(* CODESYS project Task1.project
   CompiledLibraryCompatibilityVersion: LeadSysStudio V3.5 SP15 Patch 4
   Title: Task1

Project tree, tasks and I/O mapping:
  Device : PMC600, Leadshine Technology Co., Ltd., order no. 600101, version 3.5.15.40
    application Application
      libraries: Standard, * (System)
      task MainTask (cyclic, interval t#4ms, priority 4, watchdog t#5000ms x 1) calls nothing
      task EtherCAT_Master_Leadshine_A (cyclic, interval 4000 µs, priority 0) calls PLC_PRG, EtherCAT_Master_Leadshine_A.EtherCAT_Task
      task SoftMotion_PlanningTask (freewheeling, priority 15) calls nothing
      program PLC_PRG [LD]
      axis group Tripod: TRAFO.Kin_Tripod_Rotary, axes Axis_3, Axis_4, Axis_5
    Device Diagnose
    Network Configuration
      LocalBus Config
    Resource Usage
    SoftMotion General Axis Pool
    High_Speed_IO_Module : High Speed IO Module, Leadshine Technology Co., Ltd., version 3.5.15.40
        unmapped channels: Genral_IO_IN, Genral_IO_Out
    EtherCAT_Master_Leadshine_A : EtherCAT Master Leadshine, Leadshine Technology Co., Ltd., version 3.5.9.50
        settings: MasterCycleTime = 4000
      PM32EC_LOCAL : PM32EC-LOCAL, Leadshine Technology Co., Ltd., order no. PM32EC-LOCAL, version Revision=16#20061010
          settings: StationAlias = 0; DC sync0 cycletime = 4000; DC sync1 cycletime = 4000
      DM3C_EC522 : DM3C-EC522(COE), Leadshine Technology Co.,Ltd., order no. DM3C-EC522, version Revision=16#00000001
          settings: StationAlias = 0; DC sync0 cycletime = 4000; DC sync1 cycletime = 4000; Number of SDO = 6; Homing method.Index = 16#6098; Homing method.Subindex = 16#00; Homing method.Value = 29; Homing method.Size = 8; Homing method.AbortIfError = FALSE; Homing method.JumpToLine = FALSE; Homing method.Line = 0; Homing method.CompleteAccess = FALSE; Homing velocity (fast).Index = 16#6099; Homing velocity (fast).Subindex = 16#01; Homing velocity (fast).Value = 1667; Homing velocity (fast).Size = 32; Homing velocity (fast).AbortIfError = FALSE; Homing velocity (fast).JumpToLine = FALSE; Homing velocity (fast).Line = 0; Homing velocity (fast).CompleteAccess = FALSE; Homing velocity (slow).Index = 16#6099; Homing velocity (slow).Subindex = 16#02; Homing velocity (slow).Value = 333; Homing velocity (slow).Size = 32; Homing velocity (slow).AbortIfError = FALSE; Homing velocity (slow).JumpToLine = FALSE; Homing velocity (slow).Line = 0; Homing velocity (slow).CompleteAccess = FALSE; Homing acceleration.Index = 16#609A; Homing acceleration.Subindex = 16#00; Homing acceleration.Value = 16667; Homing acceleration.Size = 32; Homing acceleration.AbortIfError = FALSE; Homing acceleration.JumpToLine = FALSE; Homing acceleration.Line = 0; Homing acceleration.CompleteAccess = FALSE; Homing offset.Index = 16#607C; Homing offset.Subindex = 16#00; Homing offset.Value = 0; Homing offset.Size = 32;
            Homing offset.AbortIfError = FALSE; Homing offset.JumpToLine = FALSE; Homing offset.Line = 0; Homing offset.CompleteAccess = FALSE
          unmapped channels: Control Word, Profile Target Position, Touch Probe Function, Last Error Code, Status Word, Modes of Operation display, Position Actual Value, Touch Probe Status, Touch Probe 1 Positive Value, Digital Inputs
        Axis : Axis, 3S - Smart Software Solutions GmbH, order no. 0, version 4.6.1.0
            settings: wDriveID = 0; dwRatioTechUnitsDenom = 500; iRatioTechUnitsNum = 3; 一圈脉冲数 = 10000; 工作台一圈的位移 = 60; 电子齿轮比分子 = 1; 电子齿轮比分母 = 1; ScalingIncs = 500; ScalingUnits = 3; AdrOffset_8010 = 4; BitOffset_8010 = 0; BitLength_8010 = 16; Address_8010 = '%QW2'; Type_8010 = 'UINT'; AddressPointer_8010 = ADR(%QW2); AdrOffset_8020 = 8; BitOffset_8020 = 0; BitLength_8020 = 32; Address_8020 = '%QD2'; Type_8020 = 'DINT'; AddressPointer_8020 = ADR(%QD2); AdrOffset_8030 = 4294967295; BitOffset_8030 = 0; BitLength_8030 = 32; Address_8030 = ''; Type_8030 = 'DINT'; AddressPointer_8030 = 0; AdrOffset_8040 = 4294967295; BitOffset_8040 = 0; BitLength_8040 = 0; Address_8040 = ''; Type_8040 = ''; AddressPointer_8040 = 0; AdrOffset_8050 = 4294967295; BitOffset_8050 = 0; BitLength_8050 = 8; Address_8050 = ''; Type_8050 = 'USINT'; AddressPointer_8050 = 0; AdrOffset_8060 = 12;
              BitOffset_8060 = 0; BitLength_8060 = 16; Address_8060 = '%QW6'; Type_8060 = 'UINT'; AddressPointer_8060 = ADR(%QW6); AdrOffset_8070 = 4294967295; BitOffset_8070 = 0; BitLength_8070 = 0; Address_8070 = ''; Type_8070 = ''; AddressPointer_8070 = 0; AdrOffset_8080 = 4294967295; BitOffset_8080 = 0; BitLength_8080 = 0; Address_8080 = ''; Type_8080 = ''; AddressPointer_8080 = 0; AdrOffset_8090 = 4294967295; BitOffset_8090 = 0; BitLength_8090 = 0; Address_8090 = ''; Type_8090 = ''; AddressPointer_8090 = 0; AdrOffset_8510 = 6; BitOffset_8510 = 0; BitLength_8510 = 16; Address_8510 = '%IW3'; Type_8510 = 'UINT'; AddressPointer_8510 = ADR(%IW3); AdrOffset_8520 = 12; BitOffset_8520 = 0; BitLength_8520 = 32; Address_8520 = '%ID3'; Type_8520 = 'DINT'; AddressPointer_8520 = ADR(%ID3); AdrOffset_8530 = 4294967295; BitOffset_8530 = 0; BitLength_8530 = 0; Address_8530 = ''; Type_8530 = '';
              AddressPointer_8530 = 0; AdrOffset_8540 = 4294967295; BitOffset_8540 = 0; BitLength_8540 = 0; Address_8540 = ''; Type_8540 = ''; AddressPointer_8540 = 0; AdrOffset_8550 = 8; BitOffset_8550 = 0; BitLength_8550 = 8; Address_8550 = '%IB8'; Type_8550 = 'SINT'; AddressPointer_8550 = ADR(%IB8); AdrOffset_8560 = 24; BitOffset_8560 = 0; BitLength_8560 = 32; Address_8560 = '%ID6'; Type_8560 = 'UDINT'; AddressPointer_8560 = ADR(%ID6); AdrOffset_8570 = 16; BitOffset_8570 = 0; BitLength_8570 = 16; Address_8570 = '%IW8'; Type_8570 = 'UINT'; AddressPointer_8570 = ADR(%IW8); AdrOffset_8580 = 20; BitOffset_8580 = 0; BitLength_8580 = 32; Address_8580 = '%ID5'; Type_8580 = 'DINT'; AddressPointer_8580 = ADR(%ID5); AdrOffset_8590 = 4294967295; BitOffset_8590 = 0; BitLength_8590 = 0; Address_8590 = ''; Type_8590 = ''; AddressPointer_8590 = 0; AdrOffset_8600 = 4294967295; BitOffset_8600 = 0; BitLength_8600 = 0;
              Address_8600 = ''; Type_8600 = ''; AddressPointer_8600 = 0; AdrOffset_8600 = 4294967295; BitOffset_8600 = 0; BitLength_8600 = 0; Address_8610 = ''; Type_8610 = ''; AddressPointer_8610 = 0; AdrOffset_8620 = 4294967295; BitOffset_8620 = 0; BitLength_8620 = 0; Address_8620 = ''; Type_8620 = ''; AddressPointer_8620 = 0
      DM3C_EC522_1 : DM3C-EC522(COE), Leadshine Technology Co.,Ltd., order no. DM3C-EC522, version Revision=16#00000001
          settings: StationAlias = 0; DC sync0 cycletime = 4000; DC sync1 cycletime = 4000; Number of SDO = 6; Homing method.Index = 16#6098; Homing method.Subindex = 16#00; Homing method.Value = 29; Homing method.Size = 8; Homing method.AbortIfError = FALSE; Homing method.JumpToLine = FALSE; Homing method.Line = 0; Homing method.CompleteAccess = FALSE; Homing velocity (fast).Index = 16#6099; Homing velocity (fast).Subindex = 16#01; Homing velocity (fast).Value = 1667; Homing velocity (fast).Size = 32; Homing velocity (fast).AbortIfError = FALSE; Homing velocity (fast).JumpToLine = FALSE; Homing velocity (fast).Line = 0; Homing velocity (fast).CompleteAccess = FALSE; Homing velocity (slow).Index = 16#6099; Homing velocity (slow).Subindex = 16#02; Homing velocity (slow).Value = 333; Homing velocity (slow).Size = 32; Homing velocity (slow).AbortIfError = FALSE; Homing velocity (slow).JumpToLine = FALSE; Homing velocity (slow).Line = 0; Homing velocity (slow).CompleteAccess = FALSE; Homing acceleration.Index = 16#609A; Homing acceleration.Subindex = 16#00; Homing acceleration.Value = 16667; Homing acceleration.Size = 32; Homing acceleration.AbortIfError = FALSE; Homing acceleration.JumpToLine = FALSE; Homing acceleration.Line = 0; Homing acceleration.CompleteAccess = FALSE; Homing offset.Index = 16#607C; Homing offset.Subindex = 16#00; Homing offset.Value = 0; Homing offset.Size = 32;
            Homing offset.AbortIfError = FALSE; Homing offset.JumpToLine = FALSE; Homing offset.Line = 0; Homing offset.CompleteAccess = FALSE
          unmapped channels: Control Word, Profile Target Position, Touch Probe Function, Last Error Code, Status Word, Modes of Operation display, Position Actual Value, Touch Probe Status, Touch Probe 1 Positive Value, Digital Inputs
        Axis_1 : Axis, 3S - Smart Software Solutions GmbH, order no. 0, version 4.6.1.0
            settings: dwRatioTechUnitsDenom = 500; iRatioTechUnitsNum = 3; 一圈脉冲数 = 10000; 工作台一圈的位移 = 60; 电子齿轮比分子 = 1; 电子齿轮比分母 = 1; ScalingIncs = 500; ScalingUnits = 3; AdrOffset_8010 = 16; BitOffset_8010 = 0; BitLength_8010 = 16; Address_8010 = '%QW8'; Type_8010 = 'UINT'; AddressPointer_8010 = ADR(%QW8); AdrOffset_8020 = 20; BitOffset_8020 = 0; BitLength_8020 = 32; Address_8020 = '%QD5'; Type_8020 = 'DINT'; AddressPointer_8020 = ADR(%QD5); AdrOffset_8030 = 4294967295; BitOffset_8030 = 0; BitLength_8030 = 32; Address_8030 = ''; Type_8030 = 'DINT'; AddressPointer_8030 = 0; AdrOffset_8040 = 4294967295; BitOffset_8040 = 0; BitLength_8040 = 0; Address_8040 = ''; Type_8040 = ''; AddressPointer_8040 = 0; AdrOffset_8050 = 4294967295; BitOffset_8050 = 0; BitLength_8050 = 8; Address_8050 = ''; Type_8050 = 'USINT'; AddressPointer_8050 = 0; AdrOffset_8060 = 24; BitOffset_8060 = 0;
              BitLength_8060 = 16; Address_8060 = '%QW12'; Type_8060 = 'UINT'; AddressPointer_8060 = ADR(%QW12); AdrOffset_8070 = 4294967295; BitOffset_8070 = 0; BitLength_8070 = 0; Address_8070 = ''; Type_8070 = ''; AddressPointer_8070 = 0; AdrOffset_8080 = 4294967295; BitOffset_8080 = 0; BitLength_8080 = 0; Address_8080 = ''; Type_8080 = ''; AddressPointer_8080 = 0; AdrOffset_8090 = 4294967295; BitOffset_8090 = 0; BitLength_8090 = 0; Address_8090 = ''; Type_8090 = ''; AddressPointer_8090 = 0; AdrOffset_8510 = 30; BitOffset_8510 = 0; BitLength_8510 = 16; Address_8510 = '%IW15'; Type_8510 = 'UINT'; AddressPointer_8510 = ADR(%IW15); AdrOffset_8520 = 36; BitOffset_8520 = 0; BitLength_8520 = 32; Address_8520 = '%ID9'; Type_8520 = 'DINT'; AddressPointer_8520 = ADR(%ID9); AdrOffset_8530 = 4294967295; BitOffset_8530 = 0; BitLength_8530 = 0; Address_8530 = ''; Type_8530 = ''; AddressPointer_8530 = 0;
              AdrOffset_8540 = 4294967295; BitOffset_8540 = 0; BitLength_8540 = 0; Address_8540 = ''; Type_8540 = ''; AddressPointer_8540 = 0; AdrOffset_8550 = 32; BitOffset_8550 = 0; BitLength_8550 = 8; Address_8550 = '%IB32'; Type_8550 = 'SINT'; AddressPointer_8550 = ADR(%IB32); AdrOffset_8560 = 48; BitOffset_8560 = 0; BitLength_8560 = 32; Address_8560 = '%ID12'; Type_8560 = 'UDINT'; AddressPointer_8560 = ADR(%ID12); AdrOffset_8570 = 40; BitOffset_8570 = 0; BitLength_8570 = 16; Address_8570 = '%IW20'; Type_8570 = 'UINT'; AddressPointer_8570 = ADR(%IW20); AdrOffset_8580 = 44; BitOffset_8580 = 0; BitLength_8580 = 32; Address_8580 = '%ID11'; Type_8580 = 'DINT'; AddressPointer_8580 = ADR(%ID11); AdrOffset_8590 = 4294967295; BitOffset_8590 = 0; BitLength_8590 = 0; Address_8590 = ''; Type_8590 = ''; AddressPointer_8590 = 0; AdrOffset_8600 = 4294967295; BitOffset_8600 = 0; BitLength_8600 = 0; Address_8600 = '';
              Type_8600 = ''; AddressPointer_8600 = 0; AdrOffset_8600 = 4294967295; BitOffset_8600 = 0; BitLength_8600 = 0; Address_8610 = ''; Type_8610 = ''; AddressPointer_8610 = 0; AdrOffset_8620 = 4294967295; BitOffset_8620 = 0; BitLength_8620 = 0; Address_8620 = ''; Type_8620 = ''; AddressPointer_8620 = 0
      DM3C_EC522_2 : DM3C-EC522(COE), Leadshine Technology Co.,Ltd., order no. DM3C-EC522, version Revision=16#00000001
          settings: StationAlias = 0; DC sync0 cycletime = 4000; DC sync1 cycletime = 4000; Number of SDO = 6; Homing method.Index = 16#6098; Homing method.Subindex = 16#00; Homing method.Value = 29; Homing method.Size = 8; Homing method.AbortIfError = FALSE; Homing method.JumpToLine = FALSE; Homing method.Line = 0; Homing method.CompleteAccess = FALSE; Homing velocity (fast).Index = 16#6099; Homing velocity (fast).Subindex = 16#01; Homing velocity (fast).Value = 25000; Homing velocity (fast).Size = 32; Homing velocity (fast).AbortIfError = FALSE; Homing velocity (fast).JumpToLine = FALSE; Homing velocity (fast).Line = 0; Homing velocity (fast).CompleteAccess = FALSE; Homing velocity (slow).Index = 16#6099; Homing velocity (slow).Subindex = 16#02; Homing velocity (slow).Value = 5000; Homing velocity (slow).Size = 32; Homing velocity (slow).AbortIfError = FALSE; Homing velocity (slow).JumpToLine = FALSE; Homing velocity (slow).Line = 0; Homing velocity (slow).CompleteAccess = FALSE; Homing acceleration.Index = 16#609A; Homing acceleration.Subindex = 16#00; Homing acceleration.Value = 250000; Homing acceleration.Size = 32; Homing acceleration.AbortIfError = FALSE; Homing acceleration.JumpToLine = FALSE; Homing acceleration.Line = 0; Homing acceleration.CompleteAccess = FALSE; Homing offset.Index = 16#607C; Homing offset.Subindex = 16#00; Homing offset.Value = 0; Homing offset.Size = 32;
            Homing offset.AbortIfError = FALSE; Homing offset.JumpToLine = FALSE; Homing offset.Line = 0; Homing offset.CompleteAccess = FALSE
          unmapped channels: Control Word, Profile Target Position, Touch Probe Function, Last Error Code, Status Word, Modes of Operation display, Position Actual Value, Touch Probe Status, Touch Probe 1 Positive Value, Digital Inputs
        Axis_2 : Axis, 3S - Smart Software Solutions GmbH, order no. 0, version 4.6.1.0
            settings: wDriveID = 2; dwRatioTechUnitsDenom = 2500; 一圈脉冲数 = 10000; 工作台一圈的位移 = 4; 电子齿轮比分子 = 1; 电子齿轮比分母 = 1; ScalingIncs = 2500; AdrOffset_8010 = 28; BitOffset_8010 = 0; BitLength_8010 = 16; Address_8010 = '%QW14'; Type_8010 = 'UINT'; AddressPointer_8010 = ADR(%QW14); AdrOffset_8020 = 32; BitOffset_8020 = 0; BitLength_8020 = 32; Address_8020 = '%QD8'; Type_8020 = 'DINT'; AddressPointer_8020 = ADR(%QD8); AdrOffset_8030 = 4294967295; BitOffset_8030 = 0; BitLength_8030 = 32; Address_8030 = ''; Type_8030 = 'DINT'; AddressPointer_8030 = 0; AdrOffset_8040 = 4294967295; BitOffset_8040 = 0; BitLength_8040 = 0; Address_8040 = ''; Type_8040 = ''; AddressPointer_8040 = 0; AdrOffset_8050 = 4294967295; BitOffset_8050 = 0; BitLength_8050 = 8; Address_8050 = ''; Type_8050 = 'USINT'; AddressPointer_8050 = 0; AdrOffset_8060 = 36; BitOffset_8060 = 0; BitLength_8060 = 16;
              Address_8060 = '%QW18'; Type_8060 = 'UINT'; AddressPointer_8060 = ADR(%QW18); AdrOffset_8070 = 4294967295; BitOffset_8070 = 0; BitLength_8070 = 0; Address_8070 = ''; Type_8070 = ''; AddressPointer_8070 = 0; AdrOffset_8080 = 4294967295; BitOffset_8080 = 0; BitLength_8080 = 0; Address_8080 = ''; Type_8080 = ''; AddressPointer_8080 = 0; AdrOffset_8090 = 4294967295; BitOffset_8090 = 0; BitLength_8090 = 0; Address_8090 = ''; Type_8090 = ''; AddressPointer_8090 = 0; AdrOffset_8510 = 54; BitOffset_8510 = 0; BitLength_8510 = 16; Address_8510 = '%IW27'; Type_8510 = 'UINT'; AddressPointer_8510 = ADR(%IW27); AdrOffset_8520 = 60; BitOffset_8520 = 0; BitLength_8520 = 32; Address_8520 = '%ID15'; Type_8520 = 'DINT'; AddressPointer_8520 = ADR(%ID15); AdrOffset_8530 = 4294967295; BitOffset_8530 = 0; BitLength_8530 = 0; Address_8530 = ''; Type_8530 = ''; AddressPointer_8530 = 0; AdrOffset_8540 = 4294967295;
              BitOffset_8540 = 0; BitLength_8540 = 0; Address_8540 = ''; Type_8540 = ''; AddressPointer_8540 = 0; AdrOffset_8550 = 56; BitOffset_8550 = 0; BitLength_8550 = 8; Address_8550 = '%IB56'; Type_8550 = 'SINT'; AddressPointer_8550 = ADR(%IB56); AdrOffset_8560 = 72; BitOffset_8560 = 0; BitLength_8560 = 32; Address_8560 = '%ID18'; Type_8560 = 'UDINT'; AddressPointer_8560 = ADR(%ID18); AdrOffset_8570 = 64; BitOffset_8570 = 0; BitLength_8570 = 16; Address_8570 = '%IW32'; Type_8570 = 'UINT'; AddressPointer_8570 = ADR(%IW32); AdrOffset_8580 = 68; BitOffset_8580 = 0; BitLength_8580 = 32; Address_8580 = '%ID17'; Type_8580 = 'DINT'; AddressPointer_8580 = ADR(%ID17); AdrOffset_8590 = 4294967295; BitOffset_8590 = 0; BitLength_8590 = 0; Address_8590 = ''; Type_8590 = ''; AddressPointer_8590 = 0; AdrOffset_8600 = 4294967295; BitOffset_8600 = 0; BitLength_8600 = 0; Address_8600 = ''; Type_8600 = '';
              AddressPointer_8600 = 0; AdrOffset_8600 = 4294967295; BitOffset_8600 = 0; BitLength_8600 = 0; Address_8610 = ''; Type_8610 = ''; AddressPointer_8610 = 0; AdrOffset_8620 = 4294967295; BitOffset_8620 = 0; BitLength_8620 = 0; Address_8620 = ''; Type_8620 = ''; AddressPointer_8620 = 0
      DM3C_EC522_3 : DM3C-EC522(COE), Leadshine Technology Co.,Ltd., order no. DM3C-EC522, version Revision=16#00000001
          settings: StationAlias = 0; DC sync0 cycletime = 4000; DC sync1 cycletime = 4000; Number of SDO = 6; Homing method.Index = 16#6098; Homing method.Subindex = 16#00; Homing method.Value = 21; Homing method.Size = 8; Homing method.AbortIfError = FALSE; Homing method.JumpToLine = FALSE; Homing method.Line = 0; Homing method.CompleteAccess = FALSE; Homing velocity (fast).Index = 16#6099; Homing velocity (fast).Subindex = 16#01; Homing velocity (fast).Value = 7500; Homing velocity (fast).Size = 32; Homing velocity (fast).AbortIfError = FALSE; Homing velocity (fast).JumpToLine = FALSE; Homing velocity (fast).Line = 0; Homing velocity (fast).CompleteAccess = FALSE; Homing velocity (slow).Index = 16#6099; Homing velocity (slow).Subindex = 16#02; Homing velocity (slow).Value = 5000; Homing velocity (slow).Size = 32; Homing velocity (slow).AbortIfError = FALSE; Homing velocity (slow).JumpToLine = FALSE; Homing velocity (slow).Line = 0; Homing velocity (slow).CompleteAccess = FALSE; Homing acceleration.Index = 16#609A; Homing acceleration.Subindex = 16#00; Homing acceleration.Value = 50000; Homing acceleration.Size = 32; Homing acceleration.AbortIfError = FALSE; Homing acceleration.JumpToLine = FALSE; Homing acceleration.Line = 0; Homing acceleration.CompleteAccess = FALSE; Homing offset.Index = 16#607C; Homing offset.Subindex = 16#00; Homing offset.Value = 0; Homing offset.Size = 32;
            Homing offset.AbortIfError = FALSE; Homing offset.JumpToLine = FALSE; Homing offset.Line = 0; Homing offset.CompleteAccess = FALSE
          unmapped channels: Control Word, Profile Target Position, Touch Probe Function, Last Error Code, Status Word, Modes of Operation display, Position Actual Value, Touch Probe Status, Touch Probe 1 Positive Value, Digital Inputs
        Axis_3 : Axis, 3S - Smart Software Solutions GmbH, order no. 0, version 4.6.1.0
            settings: wDriveID = 3; dwRatioTechUnitsDenom = 500; iRatioTechUnitsNum = -1; 一圈脉冲数 = 36000; 工作台一圈的位移 = 360; 电子齿轮比分子 = 5; 电子齿轮比分母 = 1; ScalingIncs = 500; InvertDirection = True; AdrOffset_8010 = 40; BitOffset_8010 = 0; BitLength_8010 = 16; Address_8010 = '%QW20'; Type_8010 = 'UINT'; AddressPointer_8010 = ADR(%QW20); AdrOffset_8020 = 44; BitOffset_8020 = 0; BitLength_8020 = 32; Address_8020 = '%QD11'; Type_8020 = 'DINT'; AddressPointer_8020 = ADR(%QD11); AdrOffset_8030 = 4294967295; BitOffset_8030 = 0; BitLength_8030 = 32; Address_8030 = ''; Type_8030 = 'DINT'; AddressPointer_8030 = 0; AdrOffset_8040 = 4294967295; BitOffset_8040 = 0; BitLength_8040 = 0; Address_8040 = ''; Type_8040 = ''; AddressPointer_8040 = 0; AdrOffset_8050 = 4294967295; BitOffset_8050 = 0; BitLength_8050 = 8; Address_8050 = ''; Type_8050 = 'USINT'; AddressPointer_8050 = 0; AdrOffset_8060 = 48;
              BitOffset_8060 = 0; BitLength_8060 = 16; Address_8060 = '%QW24'; Type_8060 = 'UINT'; AddressPointer_8060 = ADR(%QW24); AdrOffset_8070 = 4294967295; BitOffset_8070 = 0; BitLength_8070 = 0; Address_8070 = ''; Type_8070 = ''; AddressPointer_8070 = 0; AdrOffset_8080 = 4294967295; BitOffset_8080 = 0; BitLength_8080 = 0; Address_8080 = ''; Type_8080 = ''; AddressPointer_8080 = 0; AdrOffset_8090 = 4294967295; BitOffset_8090 = 0; BitLength_8090 = 0; Address_8090 = ''; Type_8090 = ''; AddressPointer_8090 = 0; AdrOffset_8510 = 78; BitOffset_8510 = 0; BitLength_8510 = 16; Address_8510 = '%IW39'; Type_8510 = 'UINT'; AddressPointer_8510 = ADR(%IW39); AdrOffset_8520 = 84; BitOffset_8520 = 0; BitLength_8520 = 32; Address_8520 = '%ID21'; Type_8520 = 'DINT'; AddressPointer_8520 = ADR(%ID21); AdrOffset_8530 = 4294967295; BitOffset_8530 = 0; BitLength_8530 = 0; Address_8530 = ''; Type_8530 = '';
              AddressPointer_8530 = 0; AdrOffset_8540 = 4294967295; BitOffset_8540 = 0; BitLength_8540 = 0; Address_8540 = ''; Type_8540 = ''; AddressPointer_8540 = 0; AdrOffset_8550 = 80; BitOffset_8550 = 0; BitLength_8550 = 8; Address_8550 = '%IB80'; Type_8550 = 'SINT'; AddressPointer_8550 = ADR(%IB80); AdrOffset_8560 = 96; BitOffset_8560 = 0; BitLength_8560 = 32; Address_8560 = '%ID24'; Type_8560 = 'UDINT'; AddressPointer_8560 = ADR(%ID24); AdrOffset_8570 = 88; BitOffset_8570 = 0; BitLength_8570 = 16; Address_8570 = '%IW44'; Type_8570 = 'UINT'; AddressPointer_8570 = ADR(%IW44); AdrOffset_8580 = 92; BitOffset_8580 = 0; BitLength_8580 = 32; Address_8580 = '%ID23'; Type_8580 = 'DINT'; AddressPointer_8580 = ADR(%ID23); AdrOffset_8590 = 4294967295; BitOffset_8590 = 0; BitLength_8590 = 0; Address_8590 = ''; Type_8590 = ''; AddressPointer_8590 = 0; AdrOffset_8600 = 4294967295; BitOffset_8600 = 0; BitLength_8600 = 0;
              Address_8600 = ''; Type_8600 = ''; AddressPointer_8600 = 0; AdrOffset_8600 = 4294967295; BitOffset_8600 = 0; BitLength_8600 = 0; Address_8610 = ''; Type_8610 = ''; AddressPointer_8610 = 0; AdrOffset_8620 = 4294967295; BitOffset_8620 = 0; BitLength_8620 = 0; Address_8620 = ''; Type_8620 = ''; AddressPointer_8620 = 0
      DM3C_EC522_4 : DM3C-EC522(COE), Leadshine Technology Co.,Ltd., order no. DM3C-EC522, version Revision=16#00000001
          settings: StationAlias = 0; DC sync0 cycletime = 4000; DC sync1 cycletime = 4000; Number of SDO = 6; Homing method.Index = 16#6098; Homing method.Subindex = 16#00; Homing method.Value = 21; Homing method.Size = 8; Homing method.AbortIfError = FALSE; Homing method.JumpToLine = FALSE; Homing method.Line = 0; Homing method.CompleteAccess = FALSE; Homing velocity (fast).Index = 16#6099; Homing velocity (fast).Subindex = 16#01; Homing velocity (fast).Value = 7500; Homing velocity (fast).Size = 32; Homing velocity (fast).AbortIfError = FALSE; Homing velocity (fast).JumpToLine = FALSE; Homing velocity (fast).Line = 0; Homing velocity (fast).CompleteAccess = FALSE; Homing velocity (slow).Index = 16#6099; Homing velocity (slow).Subindex = 16#02; Homing velocity (slow).Value = 5000; Homing velocity (slow).Size = 32; Homing velocity (slow).AbortIfError = FALSE; Homing velocity (slow).JumpToLine = FALSE; Homing velocity (slow).Line = 0; Homing velocity (slow).CompleteAccess = FALSE; Homing acceleration.Index = 16#609A; Homing acceleration.Subindex = 16#00; Homing acceleration.Value = 50000; Homing acceleration.Size = 32; Homing acceleration.AbortIfError = FALSE; Homing acceleration.JumpToLine = FALSE; Homing acceleration.Line = 0; Homing acceleration.CompleteAccess = FALSE; Homing offset.Index = 16#607C; Homing offset.Subindex = 16#00; Homing offset.Value = 0; Homing offset.Size = 32;
            Homing offset.AbortIfError = FALSE; Homing offset.JumpToLine = FALSE; Homing offset.Line = 0; Homing offset.CompleteAccess = FALSE
          unmapped channels: Control Word, Profile Target Position, Touch Probe Function, Last Error Code, Status Word, Modes of Operation display, Position Actual Value, Touch Probe Status, Touch Probe 1 Positive Value, Digital Inputs
        Axis_4 : Axis, 3S - Smart Software Solutions GmbH, order no. 0, version 4.6.1.0
            settings: wDriveID = 4; dwRatioTechUnitsDenom = 500; iRatioTechUnitsNum = -1; 一圈脉冲数 = 36000; 工作台一圈的位移 = 360; 电子齿轮比分子 = 5; 电子齿轮比分母 = 1; ScalingIncs = 500; InvertDirection = True; AdrOffset_8010 = 52; BitOffset_8010 = 0; BitLength_8010 = 16; Address_8010 = '%QW26'; Type_8010 = 'UINT'; AddressPointer_8010 = ADR(%QW26); AdrOffset_8020 = 56; BitOffset_8020 = 0; BitLength_8020 = 32; Address_8020 = '%QD14'; Type_8020 = 'DINT'; AddressPointer_8020 = ADR(%QD14); AdrOffset_8030 = 4294967295; BitOffset_8030 = 0; BitLength_8030 = 32; Address_8030 = ''; Type_8030 = 'DINT'; AddressPointer_8030 = 0; AdrOffset_8040 = 4294967295; BitOffset_8040 = 0; BitLength_8040 = 0; Address_8040 = ''; Type_8040 = ''; AddressPointer_8040 = 0; AdrOffset_8050 = 4294967295; BitOffset_8050 = 0; BitLength_8050 = 8; Address_8050 = ''; Type_8050 = 'USINT'; AddressPointer_8050 = 0; AdrOffset_8060 = 60;
              BitOffset_8060 = 0; BitLength_8060 = 16; Address_8060 = '%QW30'; Type_8060 = 'UINT'; AddressPointer_8060 = ADR(%QW30); AdrOffset_8070 = 4294967295; BitOffset_8070 = 0; BitLength_8070 = 0; Address_8070 = ''; Type_8070 = ''; AddressPointer_8070 = 0; AdrOffset_8080 = 4294967295; BitOffset_8080 = 0; BitLength_8080 = 0; Address_8080 = ''; Type_8080 = ''; AddressPointer_8080 = 0; AdrOffset_8090 = 4294967295; BitOffset_8090 = 0; BitLength_8090 = 0; Address_8090 = ''; Type_8090 = ''; AddressPointer_8090 = 0; AdrOffset_8510 = 102; BitOffset_8510 = 0; BitLength_8510 = 16; Address_8510 = '%IW51'; Type_8510 = 'UINT'; AddressPointer_8510 = ADR(%IW51); AdrOffset_8520 = 108; BitOffset_8520 = 0; BitLength_8520 = 32; Address_8520 = '%ID27'; Type_8520 = 'DINT'; AddressPointer_8520 = ADR(%ID27); AdrOffset_8530 = 4294967295; BitOffset_8530 = 0; BitLength_8530 = 0; Address_8530 = ''; Type_8530 = '';
              AddressPointer_8530 = 0; AdrOffset_8540 = 4294967295; BitOffset_8540 = 0; BitLength_8540 = 0; Address_8540 = ''; Type_8540 = ''; AddressPointer_8540 = 0; AdrOffset_8550 = 104; BitOffset_8550 = 0; BitLength_8550 = 8; Address_8550 = '%IB104'; Type_8550 = 'SINT'; AddressPointer_8550 = ADR(%IB104); AdrOffset_8560 = 120; BitOffset_8560 = 0; BitLength_8560 = 32; Address_8560 = '%ID30'; Type_8560 = 'UDINT'; AddressPointer_8560 = ADR(%ID30); AdrOffset_8570 = 112; BitOffset_8570 = 0; BitLength_8570 = 16; Address_8570 = '%IW56'; Type_8570 = 'UINT'; AddressPointer_8570 = ADR(%IW56); AdrOffset_8580 = 116; BitOffset_8580 = 0; BitLength_8580 = 32; Address_8580 = '%ID29'; Type_8580 = 'DINT'; AddressPointer_8580 = ADR(%ID29); AdrOffset_8590 = 4294967295; BitOffset_8590 = 0; BitLength_8590 = 0; Address_8590 = ''; Type_8590 = ''; AddressPointer_8590 = 0; AdrOffset_8600 = 4294967295; BitOffset_8600 = 0; BitLength_8600 = 0;
              Address_8600 = ''; Type_8600 = ''; AddressPointer_8600 = 0; AdrOffset_8600 = 4294967295; BitOffset_8600 = 0; BitLength_8600 = 0; Address_8610 = ''; Type_8610 = ''; AddressPointer_8610 = 0; AdrOffset_8620 = 4294967295; BitOffset_8620 = 0; BitLength_8620 = 0; Address_8620 = ''; Type_8620 = ''; AddressPointer_8620 = 0
      DM3C_EC522_5 : DM3C-EC522(COE), Leadshine Technology Co.,Ltd., order no. DM3C-EC522, version Revision=16#00000001
          settings: StationAlias = 0; DC sync0 cycletime = 4000; DC sync1 cycletime = 4000; Number of SDO = 6; Homing method.Index = 16#6098; Homing method.Subindex = 16#00; Homing method.Value = 21; Homing method.Size = 8; Homing method.AbortIfError = FALSE; Homing method.JumpToLine = FALSE; Homing method.Line = 0; Homing method.CompleteAccess = FALSE; Homing velocity (fast).Index = 16#6099; Homing velocity (fast).Subindex = 16#01; Homing velocity (fast).Value = 7500; Homing velocity (fast).Size = 32; Homing velocity (fast).AbortIfError = FALSE; Homing velocity (fast).JumpToLine = FALSE; Homing velocity (fast).Line = 0; Homing velocity (fast).CompleteAccess = FALSE; Homing velocity (slow).Index = 16#6099; Homing velocity (slow).Subindex = 16#02; Homing velocity (slow).Value = 5000; Homing velocity (slow).Size = 32; Homing velocity (slow).AbortIfError = FALSE; Homing velocity (slow).JumpToLine = FALSE; Homing velocity (slow).Line = 0; Homing velocity (slow).CompleteAccess = FALSE; Homing acceleration.Index = 16#609A; Homing acceleration.Subindex = 16#00; Homing acceleration.Value = 50000; Homing acceleration.Size = 32; Homing acceleration.AbortIfError = FALSE; Homing acceleration.JumpToLine = FALSE; Homing acceleration.Line = 0; Homing acceleration.CompleteAccess = FALSE; Homing offset.Index = 16#607C; Homing offset.Subindex = 16#00; Homing offset.Value = 0; Homing offset.Size = 32;
            Homing offset.AbortIfError = FALSE; Homing offset.JumpToLine = FALSE; Homing offset.Line = 0; Homing offset.CompleteAccess = FALSE
          unmapped channels: Control Word, Profile Target Position, Touch Probe Function, Last Error Code, Status Word, Modes of Operation display, Position Actual Value, Touch Probe Status, Touch Probe 1 Positive Value, Digital Inputs
        Axis_5 : Axis, 3S - Smart Software Solutions GmbH, order no. 0, version 4.6.1.0
            settings: wDriveID = 5; dwRatioTechUnitsDenom = 500; iRatioTechUnitsNum = -1; 一圈脉冲数 = 36000; 工作台一圈的位移 = 360; 电子齿轮比分子 = 5; 电子齿轮比分母 = 1; ScalingIncs = 500; InvertDirection = True; AdrOffset_8010 = 64; BitOffset_8010 = 0; BitLength_8010 = 16; Address_8010 = '%QW32'; Type_8010 = 'UINT'; AddressPointer_8010 = ADR(%QW32); AdrOffset_8020 = 68; BitOffset_8020 = 0; BitLength_8020 = 32; Address_8020 = '%QD17'; Type_8020 = 'DINT'; AddressPointer_8020 = ADR(%QD17); AdrOffset_8030 = 4294967295; BitOffset_8030 = 0; BitLength_8030 = 32; Address_8030 = ''; Type_8030 = 'DINT'; AddressPointer_8030 = 0; AdrOffset_8040 = 4294967295; BitOffset_8040 = 0; BitLength_8040 = 0; Address_8040 = ''; Type_8040 = ''; AddressPointer_8040 = 0; AdrOffset_8050 = 4294967295; BitOffset_8050 = 0; BitLength_8050 = 8; Address_8050 = ''; Type_8050 = 'USINT'; AddressPointer_8050 = 0; AdrOffset_8060 = 72;
              BitOffset_8060 = 0; BitLength_8060 = 16; Address_8060 = '%QW36'; Type_8060 = 'UINT'; AddressPointer_8060 = ADR(%QW36); AdrOffset_8070 = 4294967295; BitOffset_8070 = 0; BitLength_8070 = 0; Address_8070 = ''; Type_8070 = ''; AddressPointer_8070 = 0; AdrOffset_8080 = 4294967295; BitOffset_8080 = 0; BitLength_8080 = 0; Address_8080 = ''; Type_8080 = ''; AddressPointer_8080 = 0; AdrOffset_8090 = 4294967295; BitOffset_8090 = 0; BitLength_8090 = 0; Address_8090 = ''; Type_8090 = ''; AddressPointer_8090 = 0; AdrOffset_8510 = 126; BitOffset_8510 = 0; BitLength_8510 = 16; Address_8510 = '%IW63'; Type_8510 = 'UINT'; AddressPointer_8510 = ADR(%IW63); AdrOffset_8520 = 132; BitOffset_8520 = 0; BitLength_8520 = 32; Address_8520 = '%ID33'; Type_8520 = 'DINT'; AddressPointer_8520 = ADR(%ID33); AdrOffset_8530 = 4294967295; BitOffset_8530 = 0; BitLength_8530 = 0; Address_8530 = ''; Type_8530 = '';
              AddressPointer_8530 = 0; AdrOffset_8540 = 4294967295; BitOffset_8540 = 0; BitLength_8540 = 0; Address_8540 = ''; Type_8540 = ''; AddressPointer_8540 = 0; AdrOffset_8550 = 128; BitOffset_8550 = 0; BitLength_8550 = 8; Address_8550 = '%IB128'; Type_8550 = 'SINT'; AddressPointer_8550 = ADR(%IB128); AdrOffset_8560 = 144; BitOffset_8560 = 0; BitLength_8560 = 32; Address_8560 = '%ID36'; Type_8560 = 'UDINT'; AddressPointer_8560 = ADR(%ID36); AdrOffset_8570 = 136; BitOffset_8570 = 0; BitLength_8570 = 16; Address_8570 = '%IW68'; Type_8570 = 'UINT'; AddressPointer_8570 = ADR(%IW68); AdrOffset_8580 = 140; BitOffset_8580 = 0; BitLength_8580 = 32; Address_8580 = '%ID35'; Type_8580 = 'DINT'; AddressPointer_8580 = ADR(%ID35); AdrOffset_8590 = 4294967295; BitOffset_8590 = 0; BitLength_8590 = 0; Address_8590 = ''; Type_8590 = ''; AddressPointer_8590 = 0; AdrOffset_8600 = 4294967295; BitOffset_8600 = 0; BitLength_8600 = 0;
              Address_8600 = ''; Type_8600 = ''; AddressPointer_8600 = 0; AdrOffset_8600 = 4294967295; BitOffset_8600 = 0; BitLength_8600 = 0; Address_8610 = ''; Type_8610 = ''; AddressPointer_8610 = 0; AdrOffset_8620 = 4294967295; BitOffset_8620 = 0; BitLength_8620 = 0; Address_8620 = ''; Type_8620 = ''; AddressPointer_8620 = 0
      L7EC_100 : L7EC-100(COE), Leadshine Technology Co.,Ltd., order no. L7EC-100, version Revision=16#00000001
          settings: StationAlias = 0; DC sync0 cycletime = 4000; DC sync1 cycletime = 4000; Number of SDO = 6; Homing method.Index = 16#6098; Homing method.Subindex = 16#00; Homing method.Value = 1; Homing method.Size = 8; Homing method.AbortIfError = FALSE; Homing method.JumpToLine = FALSE; Homing method.Line = 0; Homing method.CompleteAccess = FALSE; Homing velocity (fast).Index = 16#6099; Homing velocity (fast).Subindex = 16#01; Homing velocity (fast).Value = 40000; Homing velocity (fast).Size = 32; Homing velocity (fast).AbortIfError = FALSE; Homing velocity (fast).JumpToLine = FALSE; Homing velocity (fast).Line = 0; Homing velocity (fast).CompleteAccess = FALSE; Homing velocity (slow).Index = 16#6099; Homing velocity (slow).Subindex = 16#02; Homing velocity (slow).Value = 8000; Homing velocity (slow).Size = 32; Homing velocity (slow).AbortIfError = FALSE; Homing velocity (slow).JumpToLine = FALSE; Homing velocity (slow).Line = 0; Homing velocity (slow).CompleteAccess = FALSE; Homing acceleration.Index = 16#609A; Homing acceleration.Subindex = 16#00; Homing acceleration.Value = 400000; Homing acceleration.Size = 32; Homing acceleration.AbortIfError = FALSE; Homing acceleration.JumpToLine = FALSE; Homing acceleration.Line = 0; Homing acceleration.CompleteAccess = FALSE; Homing offset.Index = 16#607C; Homing offset.Subindex = 16#00; Homing offset.Value = 0; Homing offset.Size = 32;
            Homing offset.AbortIfError = FALSE; Homing offset.JumpToLine = FALSE; Homing offset.Line = 0; Homing offset.CompleteAccess = FALSE
          unmapped channels: Control word, Profile target position, Touch Probe Function, Last error code, Status word, Modes of operation display, Actual motor position, Touch Probe Status, Touch probe pos1 pos value, Digital inputs
        Axis_6 : Axis, 3S - Smart Software Solutions GmbH, order no. 0, version 4.6.1.0
            settings: wDriveID = 6; dwRatioTechUnitsDenom = 4000; 一圈脉冲数 = 10000; 工作台一圈的位移 = 2.5; 电子齿轮比分子 = 1; 电子齿轮比分母 = 1; ScalingIncs = 4000; AdrOffset_8010 = 76; BitOffset_8010 = 0; BitLength_8010 = 16; Address_8010 = '%QW38'; Type_8010 = 'UINT'; AddressPointer_8010 = ADR(%QW38); AdrOffset_8020 = 80; BitOffset_8020 = 0; BitLength_8020 = 32; Address_8020 = '%QD20'; Type_8020 = 'DINT'; AddressPointer_8020 = ADR(%QD20); AdrOffset_8030 = 4294967295; BitOffset_8030 = 0; BitLength_8030 = 32; Address_8030 = ''; Type_8030 = 'DINT'; AddressPointer_8030 = 0; AdrOffset_8040 = 4294967295; BitOffset_8040 = 0; BitLength_8040 = 16; Address_8040 = ''; Type_8040 = 'INT'; AddressPointer_8040 = 0; AdrOffset_8050 = 4294967295; BitOffset_8050 = 0; BitLength_8050 = 8; Address_8050 = ''; Type_8050 = 'USINT'; AddressPointer_8050 = 0; AdrOffset_8060 = 84; BitOffset_8060 = 0; BitLength_8060 = 16;
              Address_8060 = '%QW42'; Type_8060 = 'UINT'; AddressPointer_8060 = ADR(%QW42); AdrOffset_8070 = 4294967295; BitOffset_8070 = 0; BitLength_8070 = 0; Address_8070 = ''; Type_8070 = ''; AddressPointer_8070 = 0; AdrOffset_8080 = 4294967295; BitOffset_8080 = 0; BitLength_8080 = 16; Address_8080 = ''; Type_8080 = 'INT'; AddressPointer_8080 = 0; AdrOffset_8090 = 4294967295; BitOffset_8090 = 0; BitLength_8090 = 0; Address_8090 = ''; Type_8090 = ''; AddressPointer_8090 = 0; AdrOffset_8510 = 150; BitOffset_8510 = 0; BitLength_8510 = 16; Address_8510 = '%IW75'; Type_8510 = 'UINT'; AddressPointer_8510 = ADR(%IW75); AdrOffset_8520 = 156; BitOffset_8520 = 0; BitLength_8520 = 32; Address_8520 = '%ID39'; Type_8520 = 'DINT'; AddressPointer_8520 = ADR(%ID39); AdrOffset_8530 = 4294967295; BitOffset_8530 = 0; BitLength_8530 = 0; Address_8530 = ''; Type_8530 = ''; AddressPointer_8530 = 0; AdrOffset_8540 = 4294967295;
              BitOffset_8540 = 0; BitLength_8540 = 0; Address_8540 = ''; Type_8540 = ''; AddressPointer_8540 = 0; AdrOffset_8550 = 152; BitOffset_8550 = 0; BitLength_8550 = 8; Address_8550 = '%IB152'; Type_8550 = 'SINT'; AddressPointer_8550 = ADR(%IB152); AdrOffset_8560 = 168; BitOffset_8560 = 0; BitLength_8560 = 32; Address_8560 = '%ID42'; Type_8560 = 'UDINT'; AddressPointer_8560 = ADR(%ID42); AdrOffset_8570 = 160; BitOffset_8570 = 0; BitLength_8570 = 16; Address_8570 = '%IW80'; Type_8570 = 'UINT'; AddressPointer_8570 = ADR(%IW80); AdrOffset_8580 = 164; BitOffset_8580 = 0; BitLength_8580 = 32; Address_8580 = '%ID41'; Type_8580 = 'DINT'; AddressPointer_8580 = ADR(%ID41); AdrOffset_8590 = 4294967295; BitOffset_8590 = 0; BitLength_8590 = 0; Address_8590 = ''; Type_8590 = ''; AddressPointer_8590 = 0; AdrOffset_8600 = 4294967295; BitOffset_8600 = 0; BitLength_8600 = 0; Address_8600 = ''; Type_8600 = '';
              AddressPointer_8600 = 0; AdrOffset_8600 = 4294967295; BitOffset_8600 = 0; BitLength_8600 = 0; Address_8610 = ''; Type_8610 = ''; AddressPointer_8610 = 0; AdrOffset_8620 = 4294967295; BitOffset_8620 = 0; BitLength_8620 = 0; Address_8620 = ''; Type_8620 = ''; AddressPointer_8620 = 0
    ModbusTCP_Slave_Device : Modbus TCP Slave, Leadshine Technology Co., Ltd., version 00.00.00.10
        settings: SlaveID = 1
*)

// Device/Application/PLC_PRG
PROGRAM PLC_PRG
VAR
	MC_Power_0: MC_Power;
	MC_Home_0: MC_Home;
	MC_Home_1: MC_Home;
	MC_Power_1: MC_Power;
	MC_Power_2: MC_Power;
	MC_Home_2: MC_Home;
	MC_Reset_0: MC_Reset;
	MC_Reset_1: MC_Reset;
	MC_Reset_2: MC_Reset;
	mc_jog_for_biaoding: MC_Jog;
	X: INT;
	X1: INT;
	Y1: INT;
	X0: INT;
	Y0: INT;
	LS_3AxisLineAbs_0: LS_3AxisLineAbs;
	POS0: ARRAY [0..2] OF LREAL;
	MC_Power_6: MC_Power;
	MC_Home_6: MC_Home;
	MC_MoveAbsolute_0: MC_MoveAbsolute;
	LS_3AxisLineAbs_1: LS_3AxisLineAbs;
	zjzq: BOOL;
	POS1: ARRAY [0..2] OF LREAL;
	zjfx: BOOL;
	MC_MoveAbsolute_1: MC_MoveAbsolute;
	MC_GroupEnable_0: MC_GroupEnable;
	SMC_GroupPower_0: SMC_GroupPower;
	MC_SetCoordinateTransform_0: MC_SetCoordinateTransform;
	mcs: MC_COORD_REF;
	MC_HOME_3: MC_Home;
	MC_HOME_4: MC_Home;
	MC_HOME_5: MC_Home;
	MC_Reset_3: MC_Reset;
	MC_Reset_4: MC_Reset;
	MC_Reset_5: MC_Reset;
	MC_Reset_6: MC_Reset;
	MC_MoveDirectAbsolute_0: MC_MoveDirectAbsolute;
	POS2: SMC_POS_REF;
	dd: BOOL;
	POS4: SMC_POS_REF;
	POS3: SMC_POS_REF;
	deltafx: BOOL;
	MC_MoveDirectAbsolute_1: MC_MoveDirectAbsolute;
	deltafx0: BOOL;
	MC_MoveDirectAbsolute_2: MC_MoveDirectAbsolute;
	ksdj1: BOOL;
	MC_Home_7: MC_Home;
	dj1: BOOL;
	LS_3AxisLineAbs_2: LS_3AxisLineAbs;
	POS5: ARRAY [0..2] OF LREAL;
	zjzq1: BOOL;
	LS_3AxisLineAbs_3: LS_3AxisLineAbs;
	zjfx1: BOOL;
	MC_MoveAbsolute_2: MC_MoveAbsolute;
	dd1: BOOL;
	MC_MoveDirectAbsolute_3: MC_MoveDirectAbsolute;
	MC_MoveDirectAbsolute_4: MC_MoveDirectAbsolute;
	deltafx01: BOOL;
	MC_MoveDirectAbsolute_5: MC_MoveDirectAbsolute;
	POS6: SMC_POS_REF;
	POS7: SMC_POS_REF;
	deltafx1: BOOL;
	MC_MoveAbsolute_3: MC_MoveAbsolute;
	ksdj2: BOOL;
	MC_Home_8: MC_Home;
	dj2: BOOL;
	LS_3AxisLineAbs_4: LS_3AxisLineAbs;
	zjzq2: BOOL;
	POS8: ARRAY [0..2] OF LREAL;
	LS_3AxisLineAbs_5: LS_3AxisLineAbs;
	zjfx2: BOOL;
	MC_MoveAbsolute_4: MC_MoveAbsolute;
	dd2: BOOL;
	MC_MoveDirectAbsolute_6: MC_MoveDirectAbsolute;
	MC_MoveDirectAbsolute_7: MC_MoveDirectAbsolute;
	POS9: SMC_POS_REF;
	deltafx02: BOOL;
	MC_MoveDirectAbsolute_8: MC_MoveDirectAbsolute;
	deltafx2: BOOL;
	POS10: SMC_POS_REF;
	MC_MoveAbsolute_5: MC_MoveAbsolute;
	ksdj3: BOOL;
	dj3: BOOL;
	MC_Home_9: MC_Home;
END_VAR

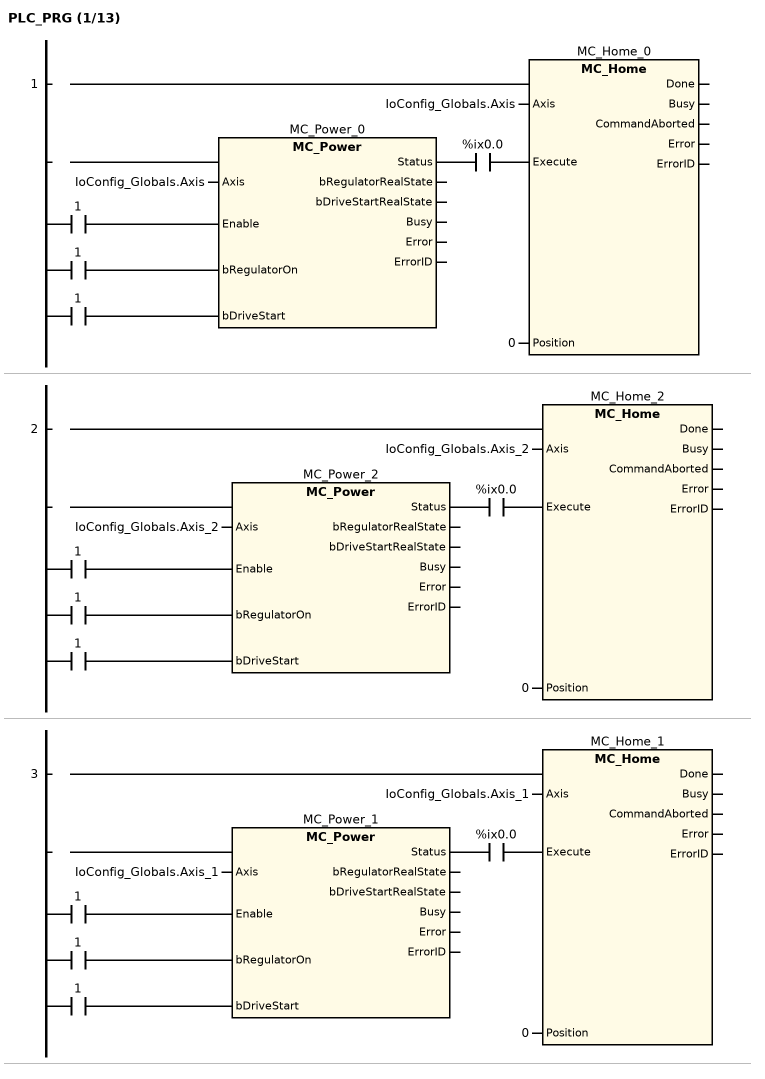
// NETWORK 1
MC_Power_0(Axis := IoConfig_Globals.Axis, Enable := 1, bRegulatorOn := 1, bDriveStart := 1); // MC_Power
MC_Home_0(Axis := IoConfig_Globals.Axis, Execute := MC_Power_0.Status AND %ix0.0, Position := 0); // MC_Home

// NETWORK 2
MC_Power_2(Axis := IoConfig_Globals.Axis_2, Enable := 1, bRegulatorOn := 1, bDriveStart := 1); // MC_Power
MC_Home_2(Axis := IoConfig_Globals.Axis_2, Execute := MC_Power_2.Status AND %ix0.0, Position := 0); // MC_Home

// NETWORK 3
MC_Power_1(Axis := IoConfig_Globals.Axis_1, Enable := 1, bRegulatorOn := 1, bDriveStart := 1); // MC_Power
MC_Home_1(Axis := IoConfig_Globals.Axis_1, Execute := MC_Power_1.Status AND %ix0.0, Position := 0); // MC_Home

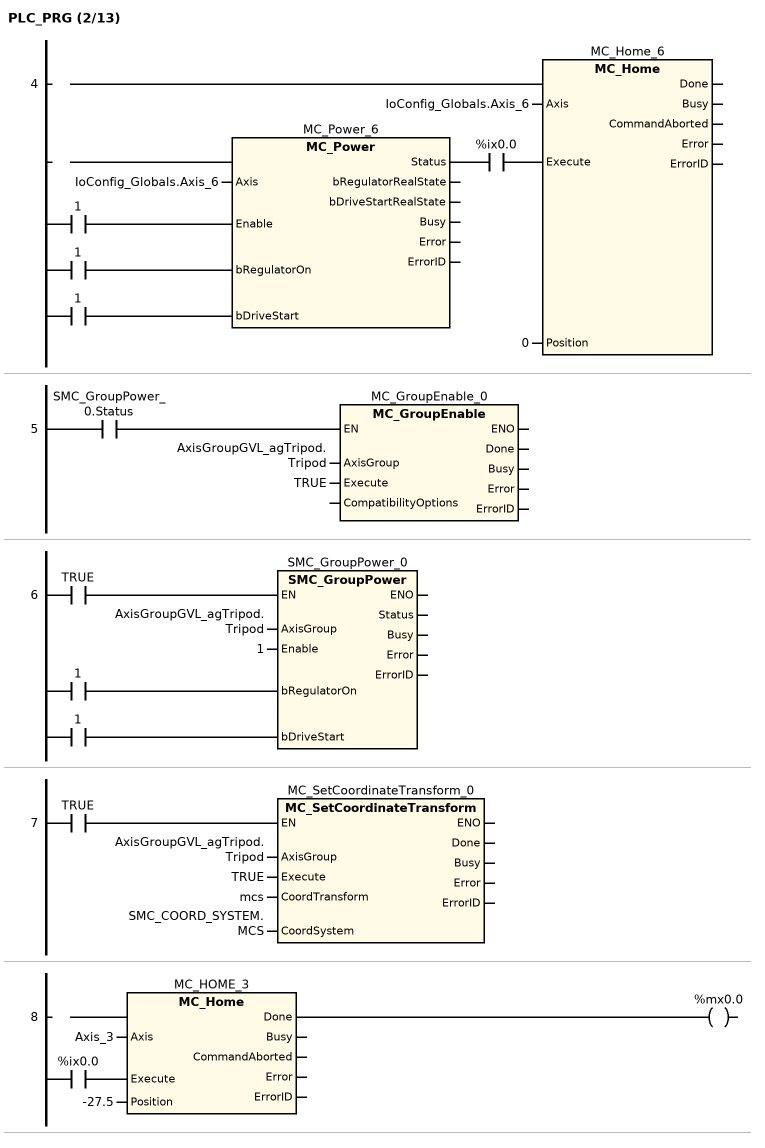
// NETWORK 4
MC_Power_6(Axis := IoConfig_Globals.Axis_6, Enable := 1, bRegulatorOn := 1, bDriveStart := 1); // MC_Power
MC_Home_6(Axis := IoConfig_Globals.Axis_6, Execute := MC_Power_6.Status AND %ix0.0, Position := 0); // MC_Home

// NETWORK 5
IF SMC_GroupPower_0.Status THEN
    MC_GroupEnable_0(AxisGroup := AxisGroupGVL_agTripod.Tripod, Execute := TRUE); // MC_GroupEnable
END_IF

// NETWORK 6
SMC_GroupPower_0(AxisGroup := AxisGroupGVL_agTripod.Tripod, Enable := 1, bRegulatorOn := 1, bDriveStart := 1); // SMC_GroupPower

// NETWORK 7
MC_SetCoordinateTransform_0(
    AxisGroup := AxisGroupGVL_agTripod.Tripod,
    Execute := TRUE,
    CoordTransform := mcs,
    CoordSystem := SMC_COORD_SYSTEM.MCS); // MC_SetCoordinateTransform

// NETWORK 8
MC_HOME_3(Axis := Axis_3, Execute := %ix0.0, Position := -27.5); // MC_Home
%mx0.0 := MC_HOME_3.Done;

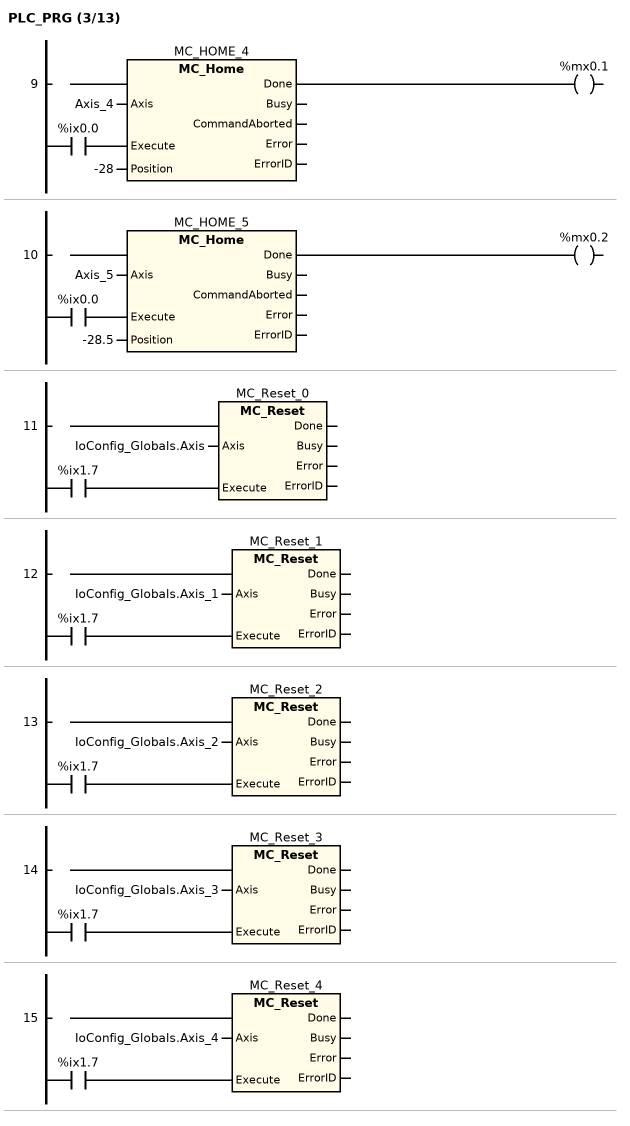
// NETWORK 9
MC_HOME_4(Axis := Axis_4, Execute := %ix0.0, Position := -28); // MC_Home
%mx0.1 := MC_HOME_4.Done;

// NETWORK 10
MC_HOME_5(Axis := Axis_5, Execute := %ix0.0, Position := -28.5); // MC_Home
%mx0.2 := MC_HOME_5.Done;

// NETWORK 11
MC_Reset_0(Axis := IoConfig_Globals.Axis, Execute := %ix1.7); // MC_Reset

// NETWORK 12
MC_Reset_1(Axis := IoConfig_Globals.Axis_1, Execute := %ix1.7); // MC_Reset

// NETWORK 13
MC_Reset_2(Axis := IoConfig_Globals.Axis_2, Execute := %ix1.7); // MC_Reset

// NETWORK 14
MC_Reset_3(Axis := IoConfig_Globals.Axis_3, Execute := %ix1.7); // MC_Reset

// NETWORK 15
MC_Reset_4(Axis := IoConfig_Globals.Axis_4, Execute := %ix1.7); // MC_Reset

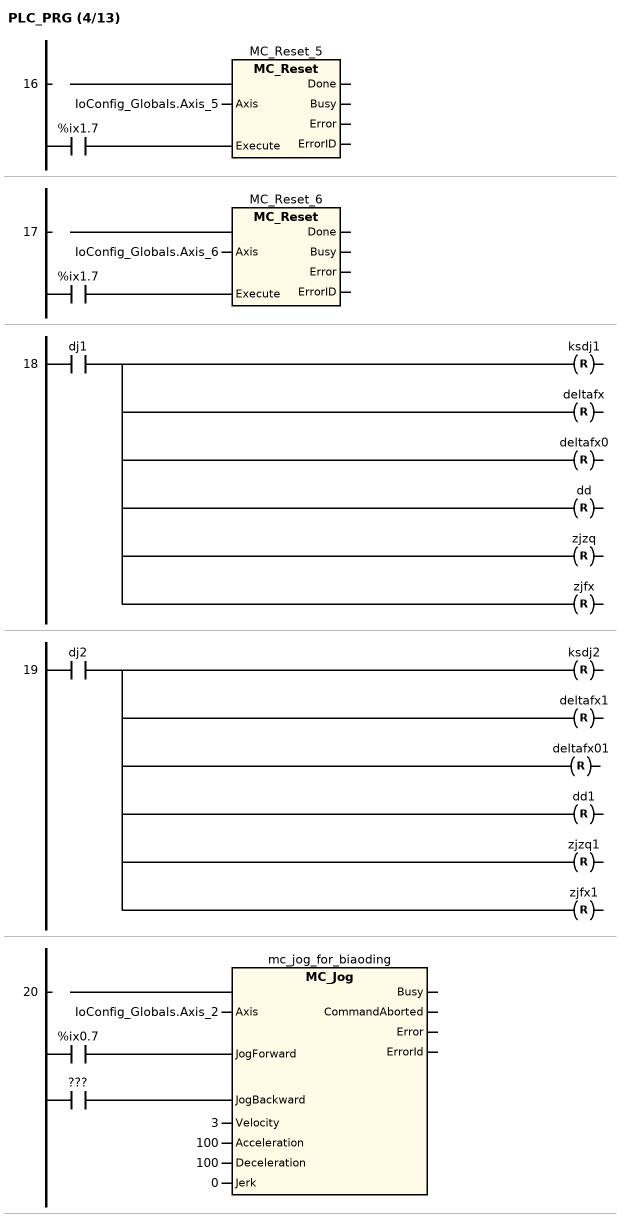
// NETWORK 16
MC_Reset_5(Axis := IoConfig_Globals.Axis_5, Execute := %ix1.7); // MC_Reset

// NETWORK 17
MC_Reset_6(Axis := IoConfig_Globals.Axis_6, Execute := %ix1.7); // MC_Reset

// NETWORK 18
ksdj1 R= dj1;
deltafx R= dj1;
deltafx0 R= dj1;
dd R= dj1;
zjzq R= dj1;
zjfx R= dj1;

// NETWORK 19
ksdj2 R= dj2;
deltafx1 R= dj2;
deltafx01 R= dj2;
dd1 R= dj2;
zjzq1 R= dj2;
zjfx1 R= dj2;

// NETWORK 20
mc_jog_for_biaoding(
    Axis := IoConfig_Globals.Axis_2,
    JogForward := %ix0.7,
    Velocity := 3,
    Acceleration := 100,
    Deceleration := 100,
    Jerk := 0); // MC_Jog

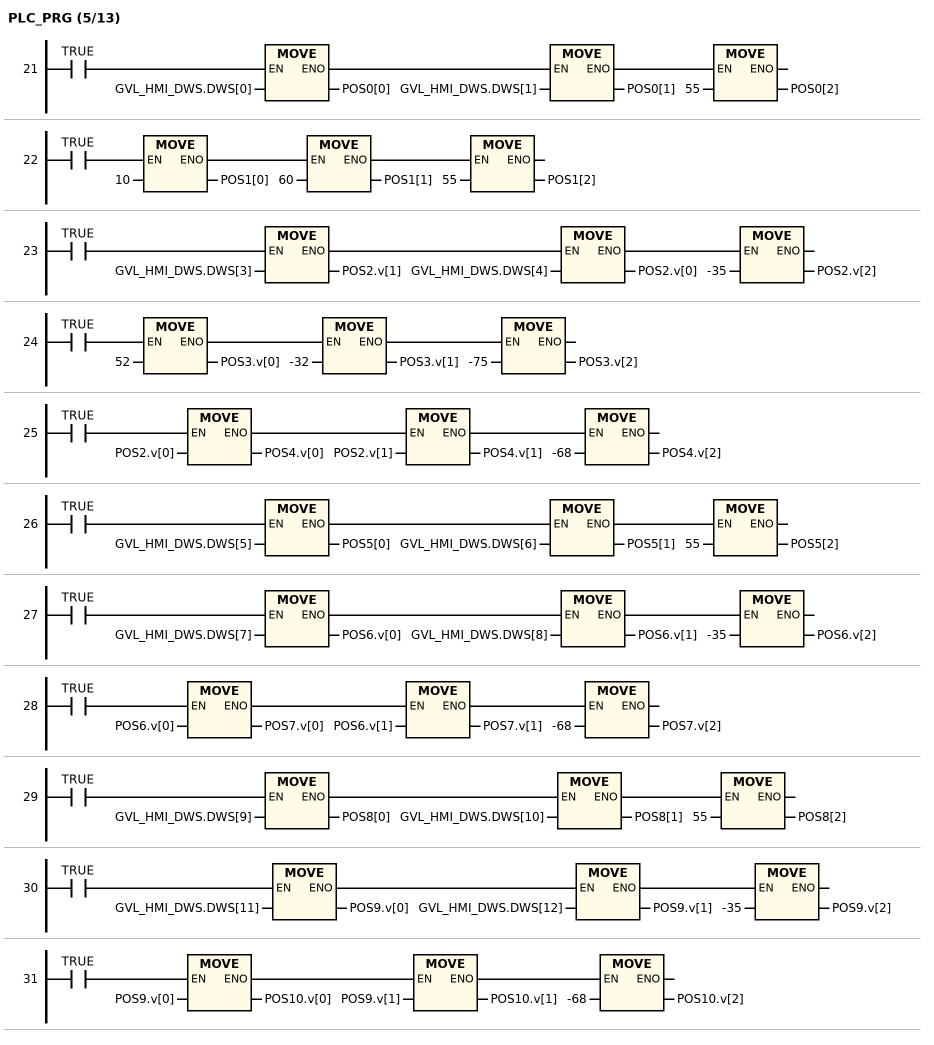
// NETWORK 21
POS0[0] := GVL_HMI_DWS.DWS[0];
POS0[1] := GVL_HMI_DWS.DWS[1];
POS0[2] := 55;

// NETWORK 22
POS1[0] := 10;
POS1[1] := 60;
POS1[2] := 55;

// NETWORK 23
POS2.v[1] := GVL_HMI_DWS.DWS[3];
POS2.v[0] := GVL_HMI_DWS.DWS[4];
POS2.v[2] := -35;

// NETWORK 24
POS3.v[0] := 52;
POS3.v[1] := -32;
POS3.v[2] := -75;

// NETWORK 25
POS4.v[0] := POS2.v[0];
POS4.v[1] := POS2.v[1];
POS4.v[2] := -68;

// NETWORK 26
POS5[0] := GVL_HMI_DWS.DWS[5];
POS5[1] := GVL_HMI_DWS.DWS[6];
POS5[2] := 55;

// NETWORK 27
POS6.v[0] := GVL_HMI_DWS.DWS[7];
POS6.v[1] := GVL_HMI_DWS.DWS[8];
POS6.v[2] := -35;

// NETWORK 28
POS7.v[0] := POS6.v[0];
POS7.v[1] := POS6.v[1];
POS7.v[2] := -68;

// NETWORK 29
POS8[0] := GVL_HMI_DWS.DWS[9];
POS8[1] := GVL_HMI_DWS.DWS[10];
POS8[2] := 55;

// NETWORK 30
POS9.v[0] := GVL_HMI_DWS.DWS[11];
POS9.v[1] := GVL_HMI_DWS.DWS[12];
POS9.v[2] := -35;

// NETWORK 31
POS10.v[0] := POS9.v[0];
POS10.v[1] := POS9.v[1];
POS10.v[2] := -68;

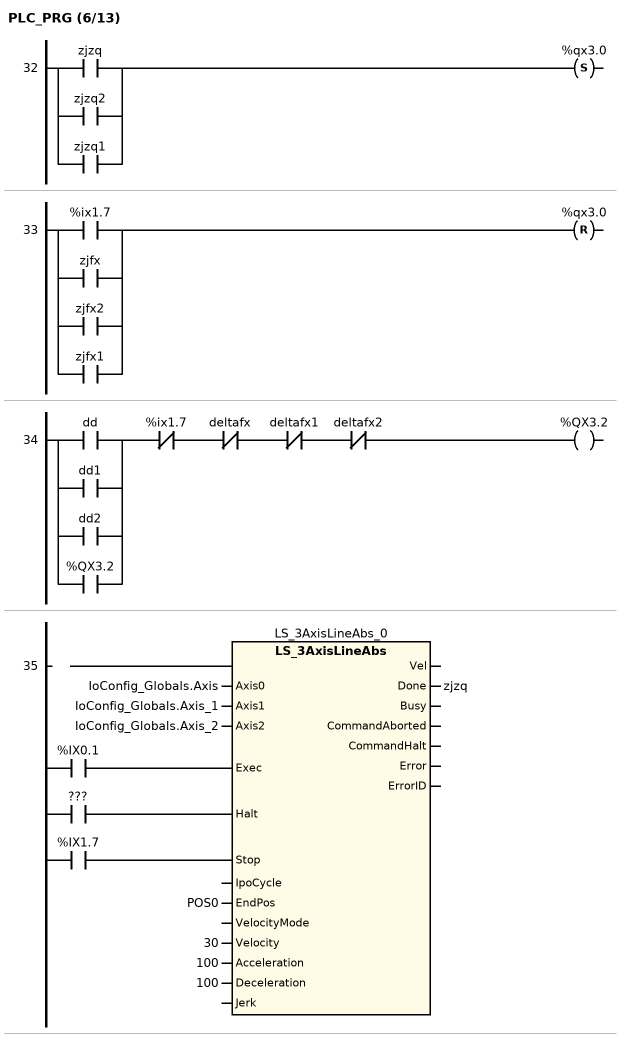
// NETWORK 32
%qx3.0 S= zjzq OR zjzq2 OR zjzq1;

// NETWORK 33
%qx3.0 R= %ix1.7 OR zjfx OR zjfx2 OR zjfx1;

// NETWORK 34
%QX3.2 := (dd OR dd1 OR dd2 OR %QX3.2) AND NOT %ix1.7 AND NOT deltafx AND NOT deltafx1 AND NOT deltafx2;

// NETWORK 35
LS_3AxisLineAbs_0(
    Axis0 := IoConfig_Globals.Axis,
    Axis1 := IoConfig_Globals.Axis_1,
    Axis2 := IoConfig_Globals.Axis_2,
    Exec := %IX0.1,
    Stop := %IX1.7,
    EndPos := POS0,
    Velocity := 30,
    Acceleration := 100,
    Deceleration := 100,
    Done => zjzq); // LS_3AxisLineAbs

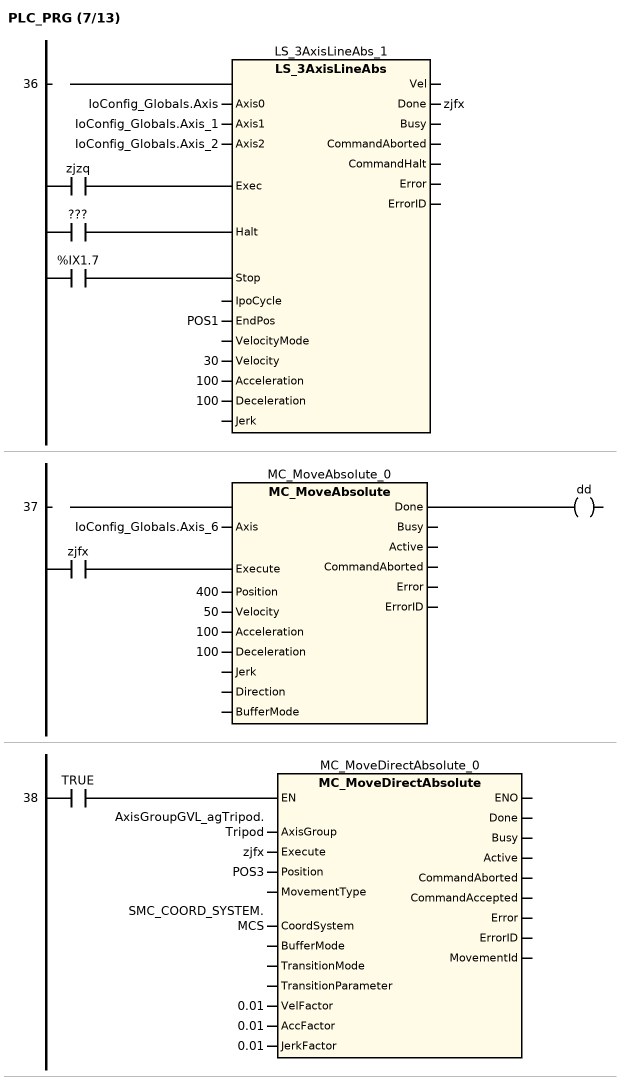
// NETWORK 36
LS_3AxisLineAbs_1(
    Axis0 := IoConfig_Globals.Axis,
    Axis1 := IoConfig_Globals.Axis_1,
    Axis2 := IoConfig_Globals.Axis_2,
    Exec := zjzq,
    Stop := %IX1.7,
    EndPos := POS1,
    Velocity := 30,
    Acceleration := 100,
    Deceleration := 100,
    Done => zjfx); // LS_3AxisLineAbs

// NETWORK 37
MC_MoveAbsolute_0(
    Axis := IoConfig_Globals.Axis_6,
    Execute := zjfx,
    Position := 400,
    Velocity := 50,
    Acceleration := 100,
    Deceleration := 100); // MC_MoveAbsolute
dd := MC_MoveAbsolute_0.Done;

// NETWORK 38
MC_MoveDirectAbsolute_0(
    AxisGroup := AxisGroupGVL_agTripod.Tripod,
    Execute := zjfx,
    Position := POS3,
    CoordSystem := SMC_COORD_SYSTEM.MCS,
    VelFactor := 0.01,
    AccFactor := 0.01,
    JerkFactor := 0.01); // MC_MoveDirectAbsolute

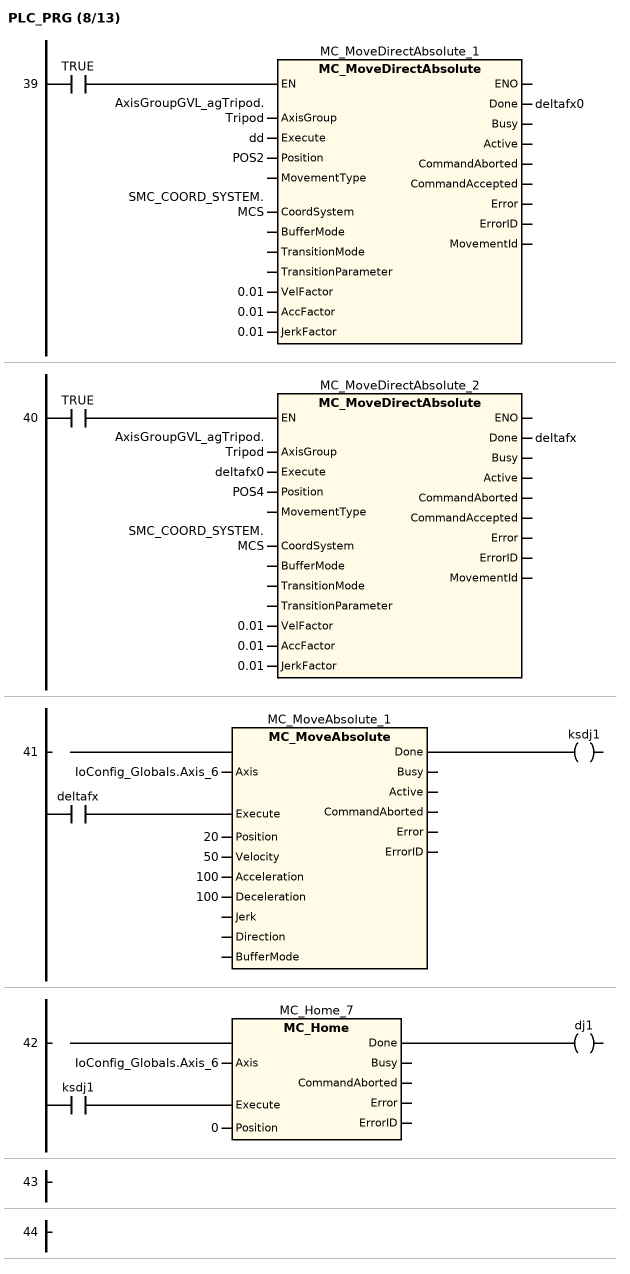
// NETWORK 39
MC_MoveDirectAbsolute_1(
    AxisGroup := AxisGroupGVL_agTripod.Tripod,
    Execute := dd,
    Position := POS2,
    CoordSystem := SMC_COORD_SYSTEM.MCS,
    VelFactor := 0.01,
    AccFactor := 0.01,
    JerkFactor := 0.01,
    Done => deltafx0); // MC_MoveDirectAbsolute

// NETWORK 40
MC_MoveDirectAbsolute_2(
    AxisGroup := AxisGroupGVL_agTripod.Tripod,
    Execute := deltafx0,
    Position := POS4,
    CoordSystem := SMC_COORD_SYSTEM.MCS,
    VelFactor := 0.01,
    AccFactor := 0.01,
    JerkFactor := 0.01,
    Done => deltafx); // MC_MoveDirectAbsolute

// NETWORK 41
MC_MoveAbsolute_1(
    Axis := IoConfig_Globals.Axis_6,
    Execute := deltafx,
    Position := 20,
    Velocity := 50,
    Acceleration := 100,
    Deceleration := 100); // MC_MoveAbsolute
ksdj1 := MC_MoveAbsolute_1.Done;

// NETWORK 42
MC_Home_7(Axis := IoConfig_Globals.Axis_6, Execute := ksdj1, Position := 0); // MC_Home
dj1 := MC_Home_7.Done;

// NETWORK 43

// NETWORK 44

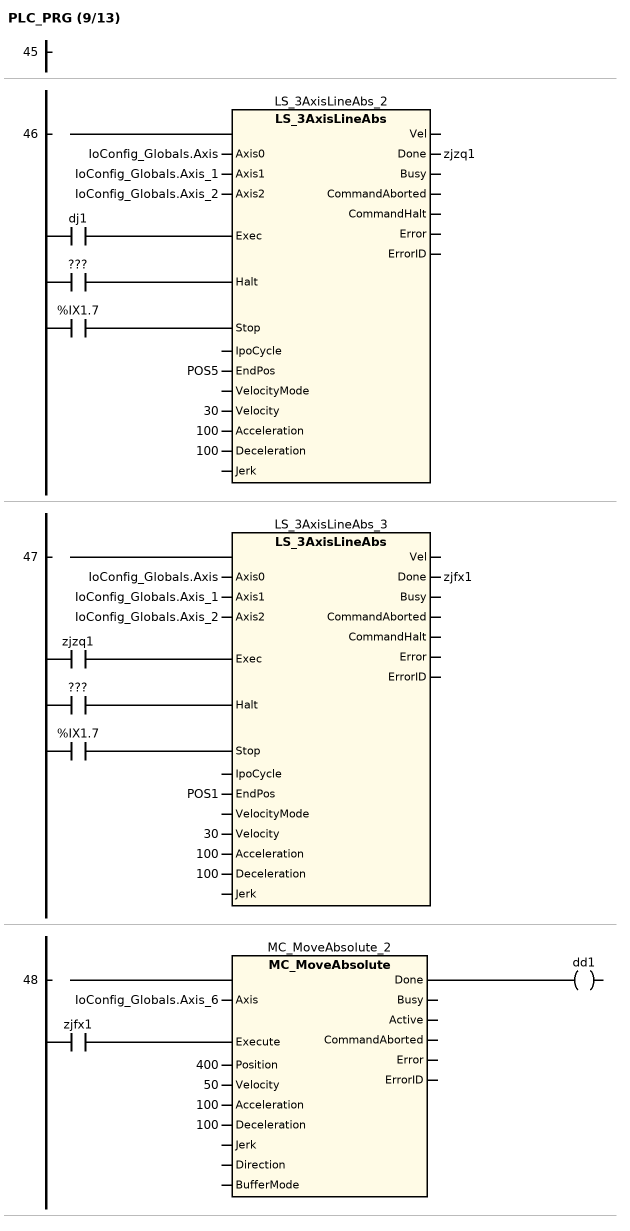
// NETWORK 45

// NETWORK 46
LS_3AxisLineAbs_2(
    Axis0 := IoConfig_Globals.Axis,
    Axis1 := IoConfig_Globals.Axis_1,
    Axis2 := IoConfig_Globals.Axis_2,
    Exec := dj1,
    Stop := %IX1.7,
    EndPos := POS5,
    Velocity := 30,
    Acceleration := 100,
    Deceleration := 100,
    Done => zjzq1); // LS_3AxisLineAbs

// NETWORK 47
LS_3AxisLineAbs_3(
    Axis0 := IoConfig_Globals.Axis,
    Axis1 := IoConfig_Globals.Axis_1,
    Axis2 := IoConfig_Globals.Axis_2,
    Exec := zjzq1,
    Stop := %IX1.7,
    EndPos := POS1,
    Velocity := 30,
    Acceleration := 100,
    Deceleration := 100,
    Done => zjfx1); // LS_3AxisLineAbs

// NETWORK 48
MC_MoveAbsolute_2(
    Axis := IoConfig_Globals.Axis_6,
    Execute := zjfx1,
    Position := 400,
    Velocity := 50,
    Acceleration := 100,
    Deceleration := 100); // MC_MoveAbsolute
dd1 := MC_MoveAbsolute_2.Done;

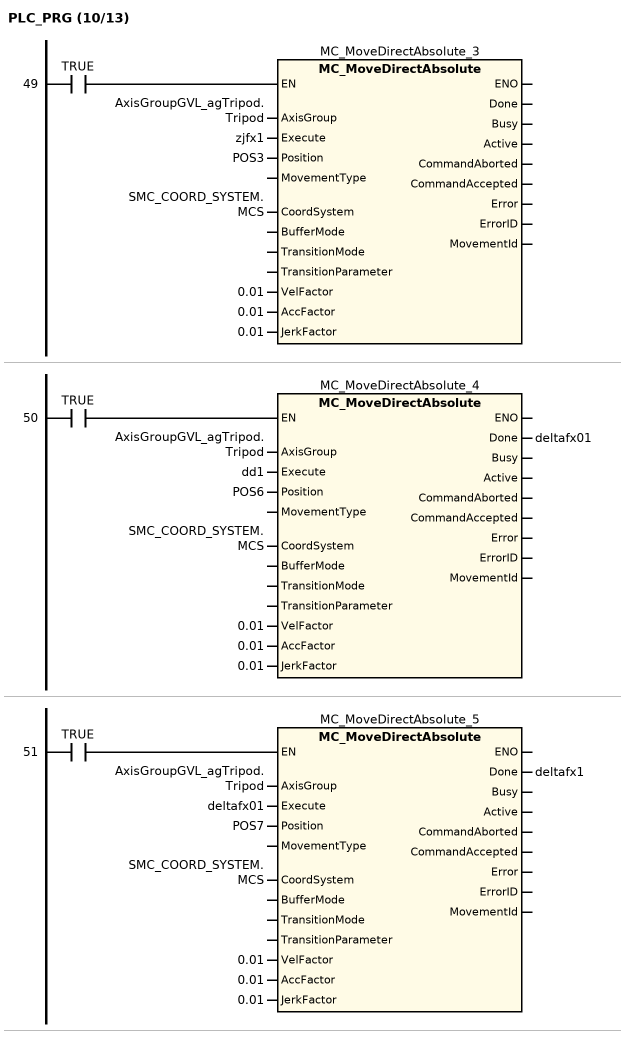
// NETWORK 49
MC_MoveDirectAbsolute_3(
    AxisGroup := AxisGroupGVL_agTripod.Tripod,
    Execute := zjfx1,
    Position := POS3,
    CoordSystem := SMC_COORD_SYSTEM.MCS,
    VelFactor := 0.01,
    AccFactor := 0.01,
    JerkFactor := 0.01); // MC_MoveDirectAbsolute

// NETWORK 50
MC_MoveDirectAbsolute_4(
    AxisGroup := AxisGroupGVL_agTripod.Tripod,
    Execute := dd1,
    Position := POS6,
    CoordSystem := SMC_COORD_SYSTEM.MCS,
    VelFactor := 0.01,
    AccFactor := 0.01,
    JerkFactor := 0.01,
    Done => deltafx01); // MC_MoveDirectAbsolute

// NETWORK 51
MC_MoveDirectAbsolute_5(
    AxisGroup := AxisGroupGVL_agTripod.Tripod,
    Execute := deltafx01,
    Position := POS7,
    CoordSystem := SMC_COORD_SYSTEM.MCS,
    VelFactor := 0.01,
    AccFactor := 0.01,
    JerkFactor := 0.01,
    Done => deltafx1); // MC_MoveDirectAbsolute

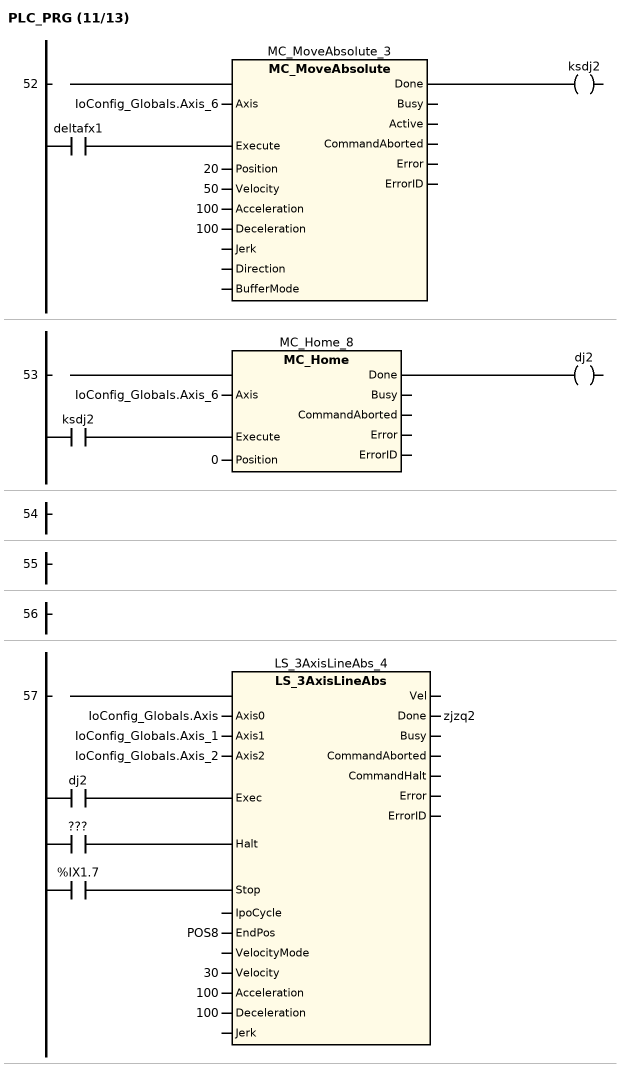
// NETWORK 52
MC_MoveAbsolute_3(
    Axis := IoConfig_Globals.Axis_6,
    Execute := deltafx1,
    Position := 20,
    Velocity := 50,
    Acceleration := 100,
    Deceleration := 100); // MC_MoveAbsolute
ksdj2 := MC_MoveAbsolute_3.Done;

// NETWORK 53
MC_Home_8(Axis := IoConfig_Globals.Axis_6, Execute := ksdj2, Position := 0); // MC_Home
dj2 := MC_Home_8.Done;

// NETWORK 54

// NETWORK 55

// NETWORK 56

// NETWORK 57
LS_3AxisLineAbs_4(
    Axis0 := IoConfig_Globals.Axis,
    Axis1 := IoConfig_Globals.Axis_1,
    Axis2 := IoConfig_Globals.Axis_2,
    Exec := dj2,
    Stop := %IX1.7,
    EndPos := POS8,
    Velocity := 30,
    Acceleration := 100,
    Deceleration := 100,
    Done => zjzq2); // LS_3AxisLineAbs

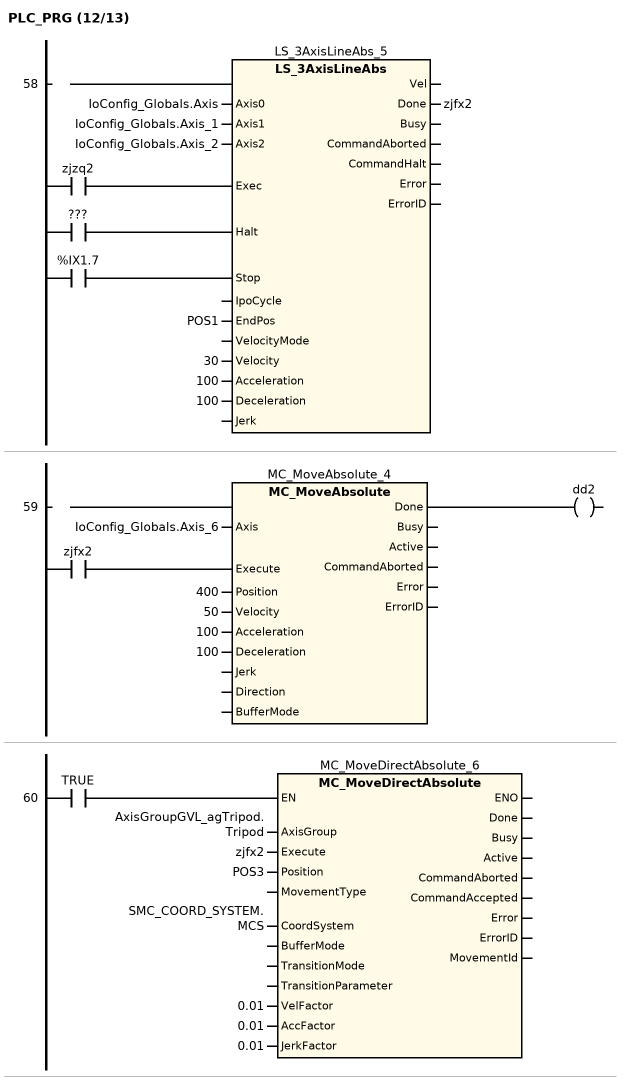
// NETWORK 58
LS_3AxisLineAbs_5(
    Axis0 := IoConfig_Globals.Axis,
    Axis1 := IoConfig_Globals.Axis_1,
    Axis2 := IoConfig_Globals.Axis_2,
    Exec := zjzq2,
    Stop := %IX1.7,
    EndPos := POS1,
    Velocity := 30,
    Acceleration := 100,
    Deceleration := 100,
    Done => zjfx2); // LS_3AxisLineAbs

// NETWORK 59
MC_MoveAbsolute_4(
    Axis := IoConfig_Globals.Axis_6,
    Execute := zjfx2,
    Position := 400,
    Velocity := 50,
    Acceleration := 100,
    Deceleration := 100); // MC_MoveAbsolute
dd2 := MC_MoveAbsolute_4.Done;

// NETWORK 60
MC_MoveDirectAbsolute_6(
    AxisGroup := AxisGroupGVL_agTripod.Tripod,
    Execute := zjfx2,
    Position := POS3,
    CoordSystem := SMC_COORD_SYSTEM.MCS,
    VelFactor := 0.01,
    AccFactor := 0.01,
    JerkFactor := 0.01); // MC_MoveDirectAbsolute

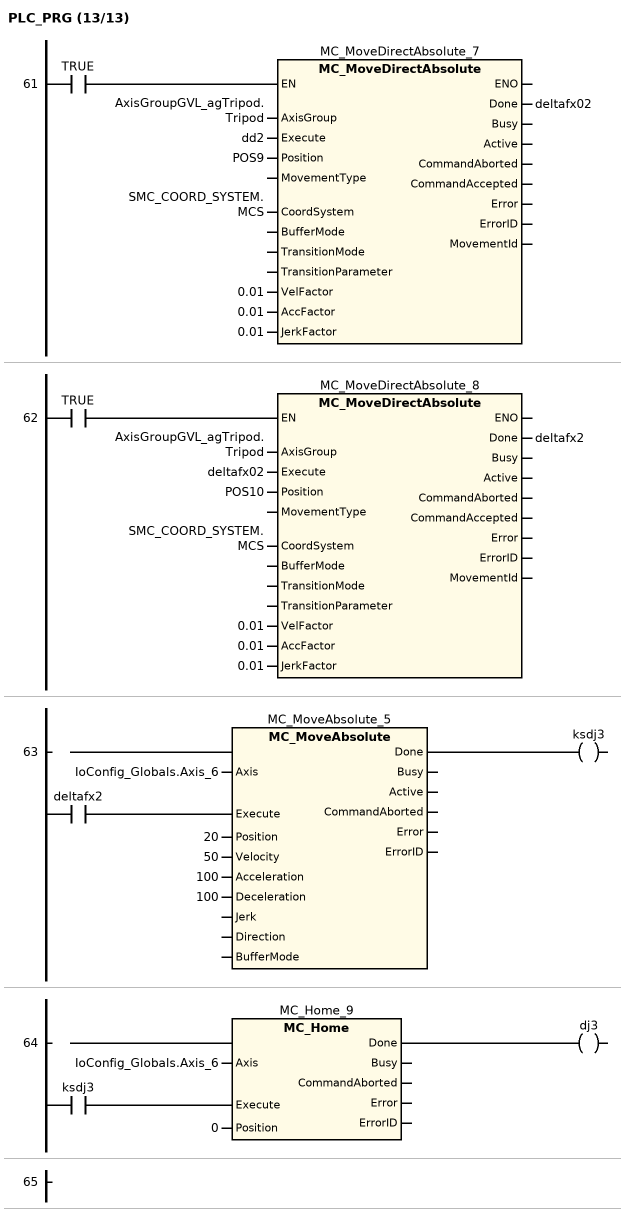
// NETWORK 61
MC_MoveDirectAbsolute_7(
    AxisGroup := AxisGroupGVL_agTripod.Tripod,
    Execute := dd2,
    Position := POS9,
    CoordSystem := SMC_COORD_SYSTEM.MCS,
    VelFactor := 0.01,
    AccFactor := 0.01,
    JerkFactor := 0.01,
    Done => deltafx02); // MC_MoveDirectAbsolute

// NETWORK 62
MC_MoveDirectAbsolute_8(
    AxisGroup := AxisGroupGVL_agTripod.Tripod,
    Execute := deltafx02,
    Position := POS10,
    CoordSystem := SMC_COORD_SYSTEM.MCS,
    VelFactor := 0.01,
    AccFactor := 0.01,
    JerkFactor := 0.01,
    Done => deltafx2); // MC_MoveDirectAbsolute

// NETWORK 63
MC_MoveAbsolute_5(
    Axis := IoConfig_Globals.Axis_6,
    Execute := deltafx2,
    Position := 20,
    Velocity := 50,
    Acceleration := 100,
    Deceleration := 100); // MC_MoveAbsolute
ksdj3 := MC_MoveAbsolute_5.Done;

// NETWORK 64
MC_Home_9(Axis := IoConfig_Globals.Axis_6, Execute := ksdj3, Position := 0); // MC_Home
dj3 := MC_Home_9.Done;

// NETWORK 65

END_PROGRAM
